Staubli VAL3: page_home_set.dtx

public string sItems
num nKey
num nIndex
public string sEvent
num nView
num nSelected
string sList
public string sMenuUser[8]
num nRefresh
num nTime = 0.5
string sMenu
bool bLarge
bool bButton[8]
num nInsert
string sMarkList
string sDataList
num nSelected1
